(* Logix 5000 project; controller OCV_Tester_EnSG vendor 1 type 14 code 106 rev 32.11; software revision 32.02 *)

TASK MainTask (continuous, watchdog 500 ms) : MainProgram

MODULES
   Local : vendor 1 type 14 code 106 (Compact 0, rev 32.11)
      DI_H2 : vendor 1 type 7 code 69 (Compact 2, rev 3.1, Input RPI 0.5 ms)
      DI_H : vendor 1 type 7 code 69 (Compact 1, rev 3.1, Input RPI 0.5 ms)
      AI : 1769-IF8 (Compact 4, rev 1.1, Output RPI 1 ms)
      DOut : vendor 1 type 7 code 73 (Compact 3, rev 3.1, Output RPI 1 ms)
      AI2 : vendor 1 type 10 code 46 (Compact 5, rev 1.1, Output RPI 1 ms)
      CPU : vendor 1 type 14 code 156 (Ethernet 172.20.7.50, rev 32.1)
      ConveyorMot : PowerFlex 525-EENET (Ethernet 172.20.9.12, rev 5.2, Output RPI 20 ms)
END_MODULES

VAR_GLOBAL   (* controller tags *)
   alwaysOK : BOOL; {constant}
   Angle : DINT := 229;
   AngleCal : DINT := 229;
   AngleOffset : DINT;
   AngleRaw : DINT := 131;   // encoder angle
   Auto : BOOL := 1;
   AVE_NOK_Control : CONTROL := (LEN := 20);
   battMon : DINT[20] := ([0] := 1552, [2] := 1641, [3] := 2222, [4] := 935, [5] := 1318, [6] := 1513, [7] := 1473, [8] := 1630, [9] := 951, [10] := 1594, [12] := 1605);
   battV : DINT[64] := ([0] := 1600, [1] := 1600, [2] := 1600, [3] := 1600, [4] := 1600, [5] := 1600, [6] := 1600, [7] := 1600, [8] := 1600, [9] := 1600, [10] := 1600, [11] := 1600, [12] := 1600, [13] := 1600, [14] := 1600, [15] := 1600, [16] := 1600, [17] := 1600, [18] := 1600, [19] := 1600, [20] := 1600, [21] := 1600, [22] := 1600, [23] := 1600, [24] := 1600, [25] := 1600, [26] := 1600, [27] := 1600, [28] := 1600, [29] := 1600, [30] := 1600, [31] := 1600, [32] := 1600, [33] := 1600, [34] := 1600, [35] := 1600, [36] := 1600, [37] := 1600, [38] := 1600, [39] := 1600, [40] := 1600, [41] := 1600, [42] := 1600, [43] := 1600, [44] := 1600, [45] := 1600, [46] := 1600, [47] := 1600, [48] := 1600, [49] := 1600, [50] := 1600, [51] := 1600, [52] := 1600, [53] := 1600, [54] := 1600, [55] := 1600, [56] := 1600, [57] := 1600, [58] := 1600, [59] := 1600,
        [60] := 1600, [61] := 1600, [62] := 1600, [63] := 1600);
   battV_NOK : INT[21] := ([0] := 1491, [1] := 1491, [2] := 1491, [3] := 1491, [4] := 1491, [5] := 1491, [6] := 1491, [7] := 1491, [8] := 1491, [9] := 1491, [10] := 1491, [11] := 1491, [12] := 1491, [13] := 1491, [14] := 1491, [15] := 1491, [16] := 1491, [17] := 1491, [18] := 1491, [19] := 1491);
   battV_NOK_avg : DINT := -25;
   blink1s : BOOL;
   blower0 : BOOL;
   cal_curVoltRaw : INT;
   cal_nom : INT := 2000; {constant}
   cal_T : DINT;
   cal_timeTOFPre : REAL := 0.25;
   cal_TimeTONPre : INT := 79;
   contact_dur_t : TIMER[20] := ([0].PRE := 2147483645, [0].ACC := 1742075, [1].PRE := 2147483645, [1].ACC := 1742075, [2].PRE := 2147483645, [2].ACC := 1742075, [3].PRE := 2147483645, [3].ACC := 1742075, [4].PRE := 2147483645, [4].ACC := 1742075, [5].PRE := 2147483645, [5].ACC := 1742075, [6].PRE := 2147483645, [6].ACC := 1742075, [7].PRE := 2147483645, [7].ACC := 1742075);
   cutOff_thrs : INT := 1597;
   d_idx : INT;
   DataV : INT[20] := ([0] := 1491, [1] := 1895, [2] := 1628, [4] := 1650, [5] := 1609, [6] := 1467, [7] := 1634, [8] := 1648, [9] := 1407, [11] := 1563, [12] := 969, [13] := 1519, [14] := 1641, [15] := 1050, [16] := 1692, [17] := 1604, [18] := 1643, [19] := 1572);
   defects : DINT[5] := ([0] := 536870911, [1] := 4324957);
   dummy3 : BOOL;
   dummy4 : BOOL;
   dummy5 : BOOL;
   eStop : BOOL;
   even : BOOL;
   fail_ejectSerp : BOOL := 1;
   fail_ejectValidation : BOOL;
   failed : BOOL[32];
   FailToRemove : BOOL := 1;   // Failed to remove battery
   Fault : BOOL;
   fault_jam : BOOL;
   FFOMonCtrl : CONTROL := (LEN := 20, POS := 19);
   FFONOKCtrl : CONTROL := (LEN := 21, POS := 20);
   FFOPrbNOKCtrl : CONTROL := (LEN := 21, POS := 20);
   FloatMode : BOOL;
   hmi_accept_thrs : INT := 1600;
   hmi_blower0 : BOOL;
   hmi_blower1 : BOOL;
   hmi_calMax : BOOL[32];
   hmi_calMin : BOOL[32];
   hmi_clearFault : BOOL;
   hmi_contactDur : DINT[20] := ([0] := 457, [1] := 1096, [2] := 2008, [3] := 182, [4] := 1187, [5] := 456, [6] := 457, [7] := 1096, [8] := 182, [9] := 273, [10] := 457, [11] := 1095, [12] := 2008, [13] := 182, [14] := 1187, [15] := 456, [16] := 457, [17] := 1096, [18] := 182, [19] := 273);   // Contact Duration
   hmi_delta : INT := 3;   // float test delta mV
   hmi_jog : BOOL;
   hmi_setSpeedRef : INT := 45;   // HMI_SetSpeed
   hmi_settingSave : BOOL;
   hmi_startingVolt : DINT := 1600;   // Init Buffer val
   i : INT;
   idx : DINT := 64;
   infeed_start_pre : INT;
   infeed_stop_pre : INT;
   lastVolt2 : DINT;
   motJam_t : DINT := 2000;   // Motor Jam T Threshold
   MotStart : BOOL;
   nc_ps_output : BOOL;
   nc_safetyContAux : BOOL;
   nofBatt : DINT := 18562;   // Number of Battery tested
   nofFailBatt : DINT := 906;
   NOK : BOOL;
   NOKK : BOOL;
   odd : BOOL;
   ons1 : DINT := 1073758208;
   Paused : BOOL;
   pb_Emergency : BOOL;
   pb_Start : BOOL;
   pb_Stop : BOOL;
   press_switch : BOOL := 1;
   probeId_NOK : INT[21] := ([0] := 1, [1] := 1, [2] := 1, [3] := 1, [4] := 1, [5] := 1, [6] := 1, [7] := 1, [8] := 1, [9] := 1, [10] := 1, [11] := 1, [12] := 1, [13] := 1, [14] := 1, [15] := 1, [16] := 1, [17] := 1, [18] := 1, [19] := 1);
   probeIdx : INT := 14;   // probe index
   ps_ejectSerp : BOOL := 1;
   ps_exist : BOOL;
   ps_index : BOOL;
   ps_inFeed : BOOL := 1;   // serpentine top
   ps_verify : BOOL;   // to verify a success remove
   ps_wheel : BOOL := 1;
   Reset : BOOL;
   Run : BOOL;
   safety_sys_ok : BOOL;
   speed : DINT;   // battery per minute
   Start : BOOL;   // Start State
   sw_door : BOOL;
   sw_doorSide : BOOL;   // Door Switch Side
   sw_doorTop : BOOL;
   timeTOFPre : DINT;
   tmr_blower0_en : BOOL;
   tmr_infeed : TIMER := (PRE := 2000);
   unloadBattV_NOK : DINT := 1491;
   unloadedBattMon : DINT := 1644;
   unloadProbe_NOK : INT := 1;
   use_calVal : BOOL;
   V_min : INT := 200;   // detect batt V
   v_rampThrs : INT := 1650;
   VMax : INT[20];
   VMin : INT[20];
   volt : INT[20];
   warning : BOOL;
   warningLamp : BOOL;
END_VAR

PROGRAM MainProgram   (* main routine MainRoutine *)
VAR
   _blower1TmrPre_tot : DINT;
   _blowerTmrPre : DINT := 130;
   _blowerTmrPre_tot : DINT := -20;
   _oddEvenRest : INT;
   AngleLimit : DINT[21] := ([0] := 340, [1] := 358, [2] := 16, [3] := 34, [4] := 52, [5] := 70, [6] := 88, [7] := 106, [8] := 124, [9] := 142, [10] := 160, [11] := 178, [12] := 196, [13] := 214, [14] := 232, [15] := 250, [16] := 268, [17] := 286, [18] := 304, [19] := 322, [20] := 340);
   AVE_Control : CONTROL := (LEN := 64);   // battery average ctrl
   battCnt : COUNTER;
   battV_avg : DINT := 1600;   // battery voltage average
   blower0_tof_pre : DINT;
   blower_react_ms : DINT := 20;
   BSLCtrl : CONTROL := (LEN := 64);
   buf_battVLen : INT := 64;   // buffer length 64
   calcSpeed : BOOL;
   clearFFO : BOOL;
   contact_Idx : INT;
   contact_t : TIMER[20] := ([0].PRE := 2147483647, [1].PRE := 2147483647, [2].PRE := 2147483647, [3].PRE := 2147483647, [4].PRE := 2147483647, [5].PRE := 2147483647, [6].PRE := 2147483647, [7].PRE := 2147483647, [8].PRE := 2147483647, [9].PRE := 2147483647, [10].PRE := 2147483647, [11].PRE := 2147483647, [12].PRE := 2147483647, [13].PRE := 2147483647, [14].PRE := 2147483647, [15].PRE := 2147483647, [16].PRE := 2147483647, [17].PRE := 2147483647, [18].PRE := 2147483647, [19].PRE := 2147483647);
   contactDur_t : TIMER[20];
   Data1 : DINT;
   dbc_tof : TIMER[2] := ([0].PRE := 2, [0].EN := 1, [0].DN := 1);
   dbc_ton : TIMER[2] := ([0].PRE := 2, [0].ACC := 3, [0].EN := 1, [0].DN := 1);
   DelayBlow : BOOL;
   deltaNofBatt : DINT;
   deltaTSpeed : DINT;
   dummyProbeEn : BOOL;
   en_blower : BOOL := 1;
   enableDummyPsIndex : BOOL;
   Failed : BOOL;
   FFOCtrl : CONTROL := (LEN := 60, POS := 60, DN := 1);
   FFOCtrl_defects : CONTROL;
   fifo : DINT;
   ForVIdx : DINT := 11;
   freeTmr : TIMER := (PRE := 2147483646, ACC := 138932, EN := 1, TT := 1);
   hmi_rev : BOOL := 1;
   hmi_setAngle0 : BOOL;   // set Offset Angle 0
   hmi_setSpeedRef100 : INT := 4500;   // hmi_setSpeedRef*100
   index : BOOL;
   lastScan : DINT := 138932;
   lastVolt : DINT;
   MaxV : INT[20] := ([1] := 1895, [2] := 1619, [3] := 1635, [4] := 1543, [5] := 1170, [8] := 287);
   nofBattOld : DINT;
   OK : BOOL := 1;
   ons : INT;
   ons2 : DINT := 68;
   Passed : BOOL;
   pb_DoorSw : BOOL;
   pb_SafetyRst : BOOL;   // pb safety reset
   ps_exist_ons : BOOL;
   px_inFeed : BOOL;   // serpentine top
   Safety : BOOL;
   StartAngle : DINT := 340;
   startContact_ts : DINT[20] := ([0] := 138649, [1] := 138887, [2] := 138808, [3] := 138887, [4] := 98255);   // Contact start
   TimeTONPre : DINT := -79;
   tmr_blower0 : TIMER := (PRE := 229);
   tmr_blower0_en : BOOL;
   tmr_blower0_TOF : TIMER := (PRE := 77);
   tmr_infeed_start : TIMER := (PRE := 1700, EN := 1, DN := 1);
   tmr_infeed_stop : TIMER := (PRE := 250);
   TmrDuration : TIMER := (PRE := 2147483647);
   tof1s : TIMER := (TT := 1, DN := 1);
   ton1s : TIMER;
   ton_blower0 : DINT;
   unloadBattV : DINT;   // unloaded battV element array
   unloadFFODefects : DINT;   // unloaded defects fifo element
END_VAR

ROUTINE _00_Diagnostics   (* ladder *)
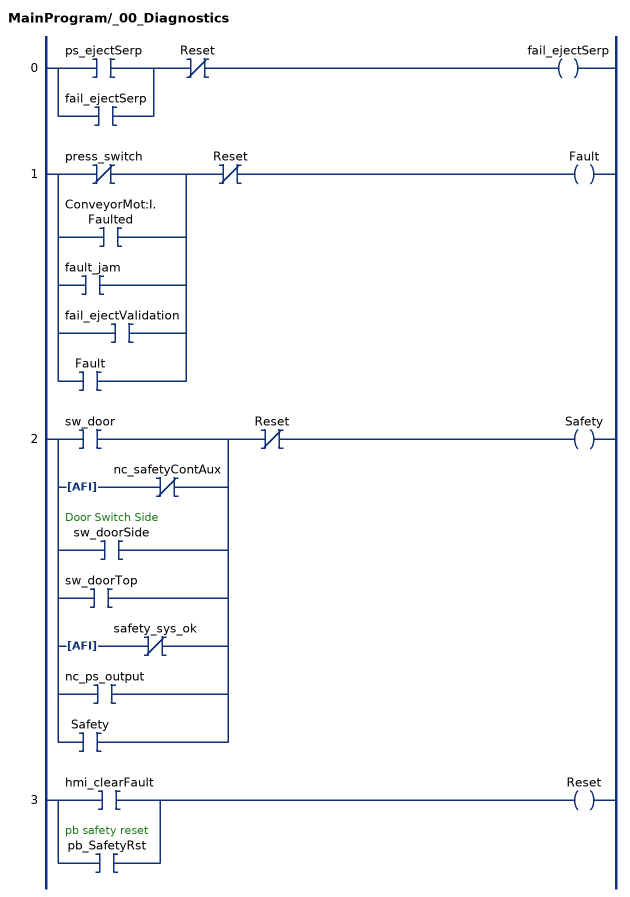
   0: [XIC(ps_ejectSerp) ,XIC(fail_ejectSerp) ]XIO(Reset)OTE(fail_ejectSerp);
   1: [XIO(press_switch) ,XIC(ConveyorMot:I.Faulted) ,XIC(fault_jam) ,XIC(fail_ejectValidation) ,XIC(Fault) ]XIO(Reset)OTE(Fault);
   2: [XIC(sw_door) ,AFI() XIO(nc_safetyContAux) ,XIC(sw_doorSide) ,XIC(sw_doorTop) ,AFI() XIO(safety_sys_ok) ,XIC(nc_ps_output) ,XIC(Safety) ]XIO(Reset)OTE(Safety);
   3: [XIC(hmi_clearFault) ,XIC(pb_SafetyRst) ]OTE(Reset);
END_ROUTINE

ROUTINE _01_Inputs   (* ladder *)
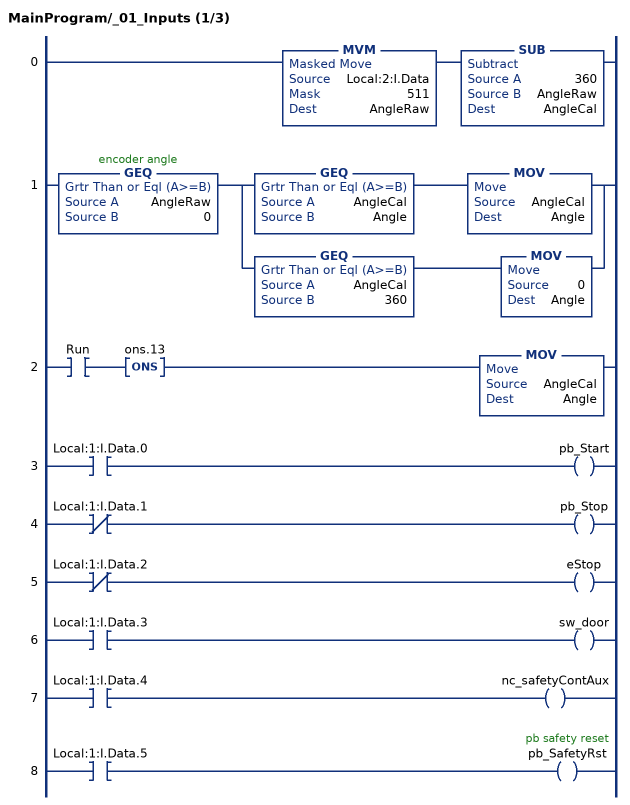
   0: MVM(Local:2:I.Data,511,AngleRaw)SUB(360,AngleRaw,AngleCal);
   1: GEQ(AngleRaw,0)[GEQ(AngleCal,Angle) MOV(AngleCal,Angle) ,GEQ(AngleCal,360) MOV(0,Angle) ];
   2: XIC(Run)ONS(ons.13)MOV(AngleCal,Angle);
   3: XIC(Local:1:I.Data.0)OTE(pb_Start);
   4: XIO(Local:1:I.Data.1)OTE(pb_Stop);
   5: XIO(Local:1:I.Data.2)OTE(eStop);
   6: XIC(Local:1:I.Data.3)OTE(sw_door);
   7: XIC(Local:1:I.Data.4)OTE(nc_safetyContAux);
   8: XIC(Local:1:I.Data.5)OTE(pb_SafetyRst);
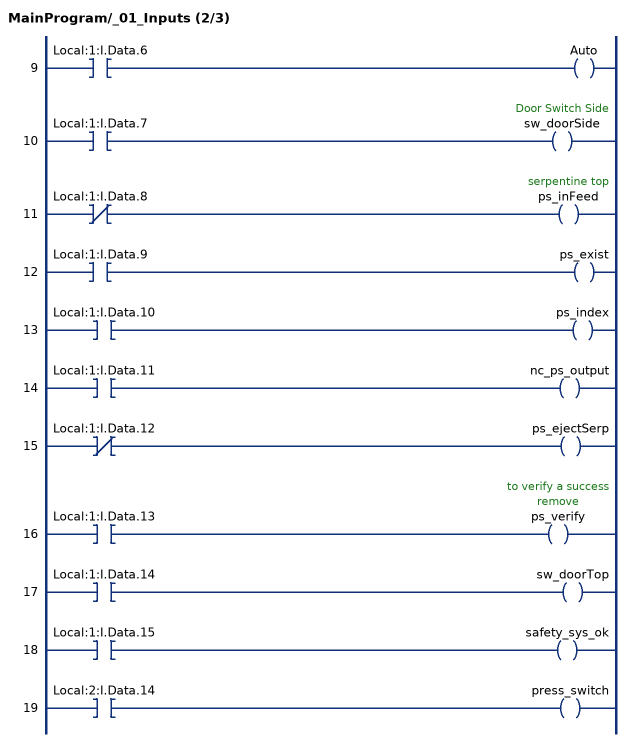
   9: XIC(Local:1:I.Data.6)OTE(Auto);
   10: XIC(Local:1:I.Data.7)OTE(sw_doorSide);
   11: XIO(Local:1:I.Data.8)OTE(ps_inFeed);
   12: XIC(Local:1:I.Data.9)OTE(ps_exist);
   13: XIC(Local:1:I.Data.10)OTE(ps_index);
   14: XIC(Local:1:I.Data.11)OTE(nc_ps_output);
   15: XIO(Local:1:I.Data.12)OTE(ps_ejectSerp);
   16: XIC(Local:1:I.Data.13)OTE(ps_verify);
   17: XIC(Local:1:I.Data.14)OTE(sw_doorTop);
   18: XIC(Local:1:I.Data.15)OTE(safety_sys_ok);
   19: XIC(Local:2:I.Data.14)OTE(press_switch);
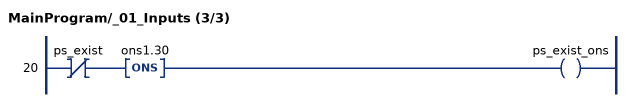
   20: XIO(ps_exist)ONS(ons1.30)OTE(ps_exist_ons);
END_ROUTINE

ROUTINE _02_Run   (* ladder *)
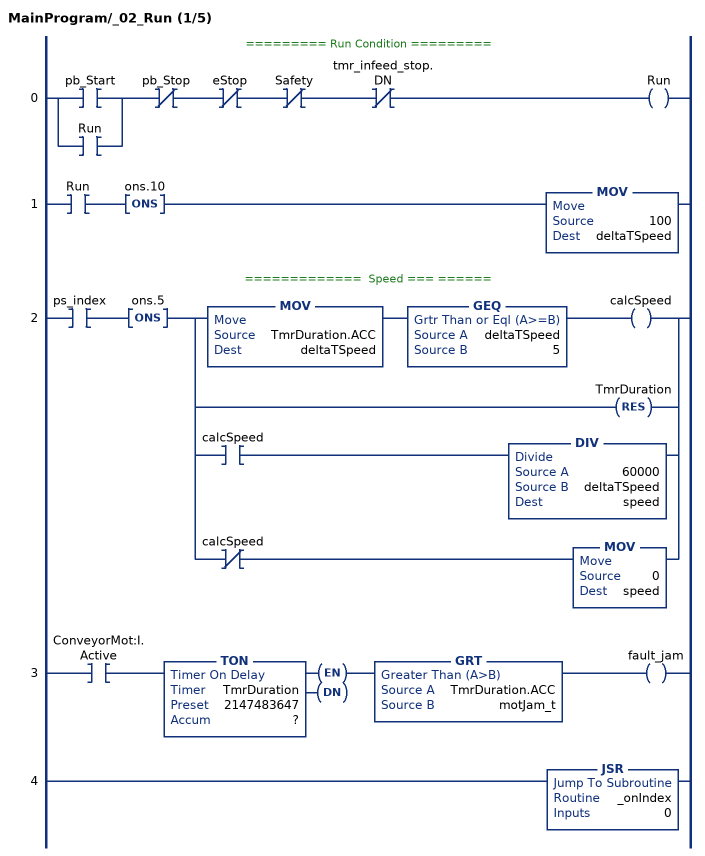
   // ========= Run Condition =========
   0: [XIC(pb_Start) ,XIC(Run) ]XIO(pb_Stop)XIO(eStop)XIO(Safety)XIO(tmr_infeed_stop.DN)OTE(Run);
   1: XIC(Run)ONS(ons.10)MOV(100,deltaTSpeed);
   // =============  Speed === ======
   2: XIC(ps_index)ONS(ons.5)[MOV(TmrDuration.ACC,deltaTSpeed) GEQ(deltaTSpeed,5) OTE(calcSpeed) ,RES(TmrDuration) ,XIC(calcSpeed) DIV(60000,deltaTSpeed,speed) ,XIO(calcSpeed) MOV(0,speed) ];
   3: XIC(ConveyorMot:I.Active)TON(TmrDuration,?,?)GRT(TmrDuration.ACC,motJam_t)OTE(fault_jam);
   4: JSR(_onIndex,0);
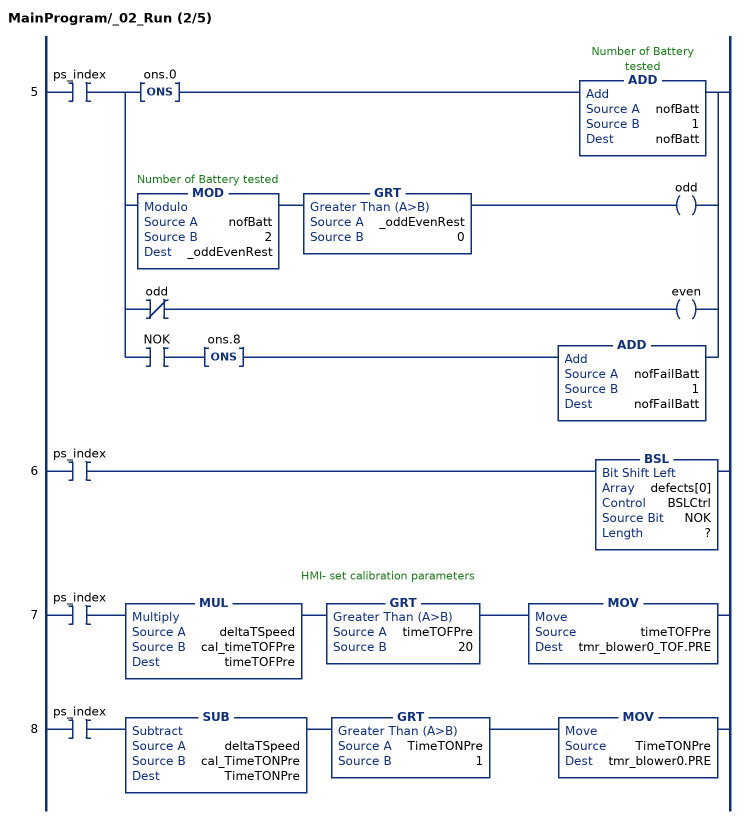
   5: XIC(ps_index)[ONS(ons.0) ADD(nofBatt,1,nofBatt) ,MOD(nofBatt,2,_oddEvenRest) GRT(_oddEvenRest,0) OTE(odd) ,XIO(odd) OTE(even) ,XIC(NOK) ONS(ons.8) ADD(nofFailBatt,1,nofFailBatt) ];
   6: XIC(ps_index)BSL(defects[0],BSLCtrl,NOK,?);
   // HMI- set calibration parameters
   7: XIC(ps_index)MUL(deltaTSpeed,cal_timeTOFPre,timeTOFPre)GRT(timeTOFPre,20)MOV(timeTOFPre,tmr_blower0_TOF.PRE);
   8: XIC(ps_index)SUB(deltaTSpeed,cal_TimeTONPre,TimeTONPre)GRT(TimeTONPre,1)MOV(TimeTONPre,tmr_blower0.PRE);
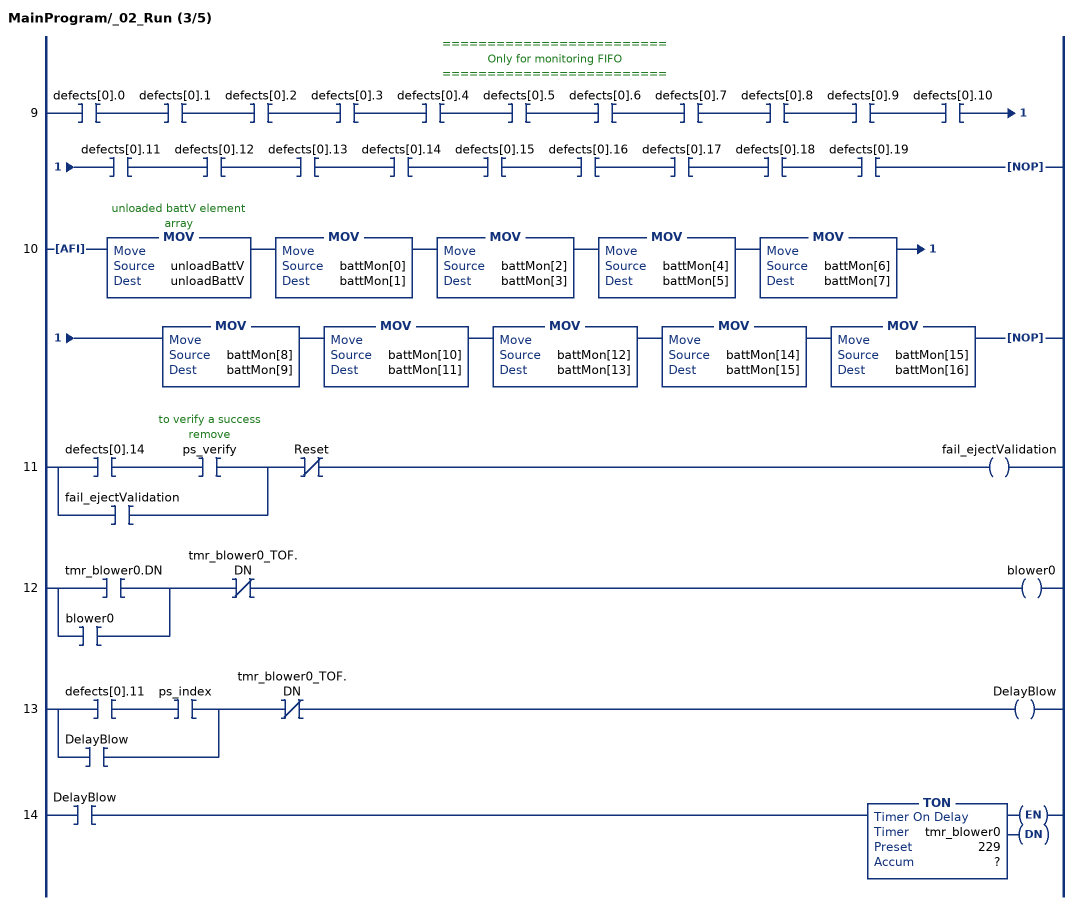
   // =========================
   // Only for monitoring FIFO
   // =========================
   9: XIC(defects[0].0)XIC(defects[0].1)XIC(defects[0].2)XIC(defects[0].3)XIC(defects[0].4)XIC(defects[0].5)XIC(defects[0].6)XIC(defects[0].7)XIC(defects[0].8)XIC(defects[0].9)XIC(defects[0].10)XIC(defects[0].11)XIC(defects[0].12)XIC(defects[0].13)XIC(defects[0].14)XIC(defects[0].15)XIC(defects[0].16)XIC(defects[0].17)XIC(defects[0].18)XIC(defects[0].19)NOP();
   10: AFI()MOV(unloadBattV,unloadBattV)MOV(battMon[0],battMon[1])MOV(battMon[2],battMon[3])MOV(battMon[4],battMon[5])MOV(battMon[6],battMon[7])MOV(battMon[8],battMon[9])MOV(battMon[10],battMon[11])MOV(battMon[12],battMon[13])MOV(battMon[14],battMon[15])MOV(battMon[15],battMon[16])NOP();
   11: [XIC(defects[0].14) XIC(ps_verify) ,XIC(fail_ejectValidation) ]XIO(Reset)OTE(fail_ejectValidation);
   12: [XIC(tmr_blower0.DN) ,XIC(blower0) ]XIO(tmr_blower0_TOF.DN)OTE(blower0);
   13: [XIC(defects[0].11) XIC(ps_index) ,XIC(DelayBlow) ]XIO(tmr_blower0_TOF.DN)OTE(DelayBlow);
   14: XIC(DelayBlow)TON(tmr_blower0,?,?);
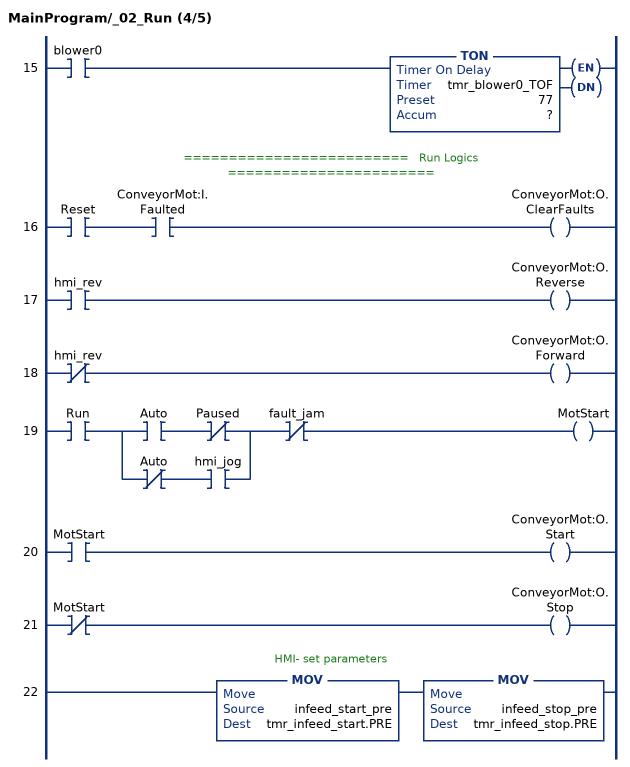
   15: XIC(blower0)TON(tmr_blower0_TOF,?,?);
   // =========================   Run Logics   =======================
   16: XIC(Reset)XIC(ConveyorMot:I.Faulted)OTE(ConveyorMot:O.ClearFaults);
   17: XIC(hmi_rev)OTE(ConveyorMot:O.Reverse);
   18: XIO(hmi_rev)OTE(ConveyorMot:O.Forward);
   19: XIC(Run)[XIC(Auto) XIO(Paused) ,XIO(Auto) XIC(hmi_jog) ]XIO(fault_jam)OTE(MotStart);
   20: XIC(MotStart)OTE(ConveyorMot:O.Start);
   21: XIO(MotStart)OTE(ConveyorMot:O.Stop);
   // HMI- set parameters
   22: MOV(infeed_start_pre,tmr_infeed_start.PRE)MOV(infeed_stop_pre,tmr_infeed_stop.PRE);
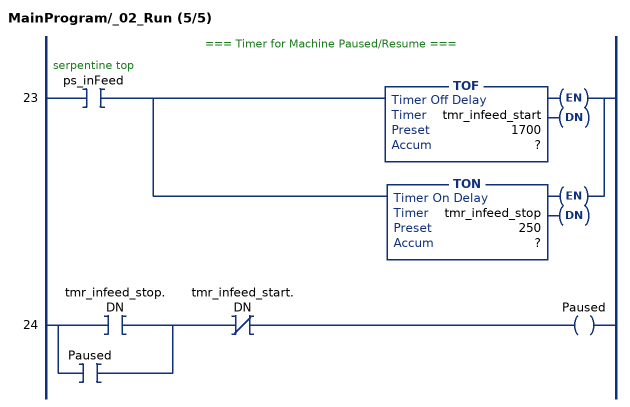
   // === Timer for Machine Paused/Resume ===
   23: XIC(ps_inFeed)[TOF(tmr_infeed_start,?,?) ,TON(tmr_infeed_stop,?,?) ];
   24: [XIC(tmr_infeed_stop.DN) ,XIC(Paused) ]XIO(tmr_infeed_start.DN)OTE(Paused);
END_ROUTINE

ROUTINE _03_Angle   (* ladder *)
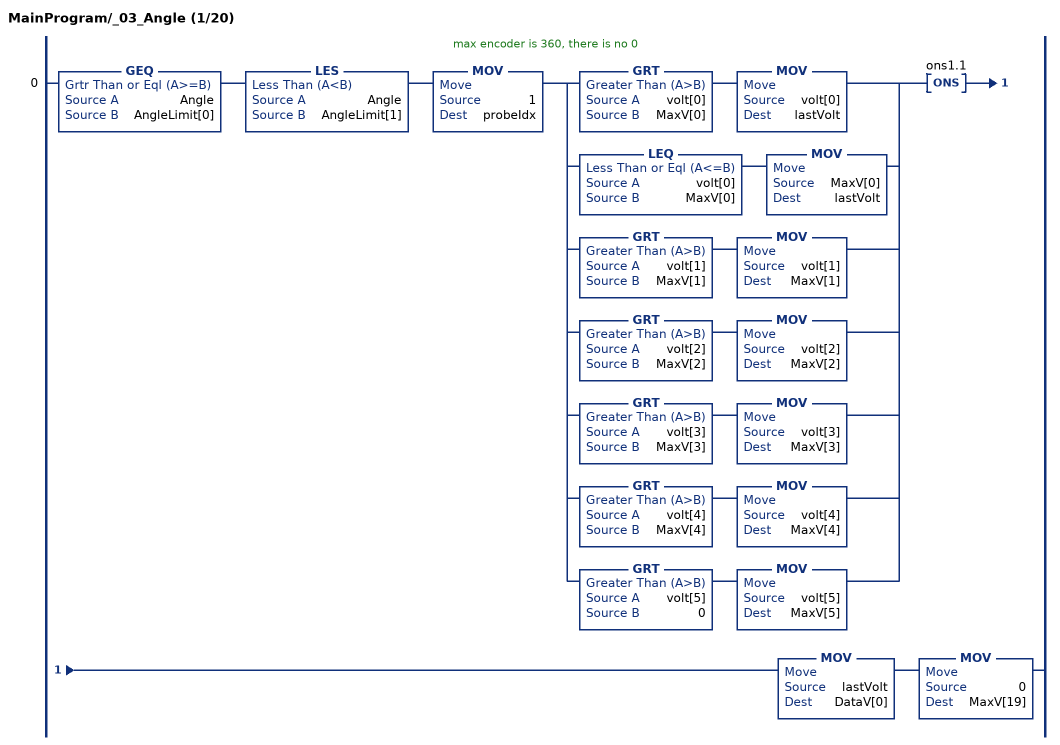
   // max encoder is 360, there is no 0
   0: GEQ(Angle,AngleLimit[0])LES(Angle,AngleLimit[1])MOV(1,probeIdx)[GRT(volt[0],MaxV[0]) MOV(volt[0],lastVolt) ,LEQ(volt[0],MaxV[0]) MOV(MaxV[0],lastVolt) ,GRT(volt[1],MaxV[1]) MOV(volt[1],MaxV[1]) ,GRT(volt[2],MaxV[2]) MOV(volt[2],MaxV[2]) ,GRT(volt[3],MaxV[3]) MOV(volt[3],MaxV[3]) ,GRT(volt[4],MaxV[4]) MOV(volt[4],MaxV[4]) ,GRT(volt[5],0) MOV(volt[5],MaxV[5]) ]ONS(ons1.1)MOV(lastVolt,DataV[0])MOV(0,MaxV[19]);
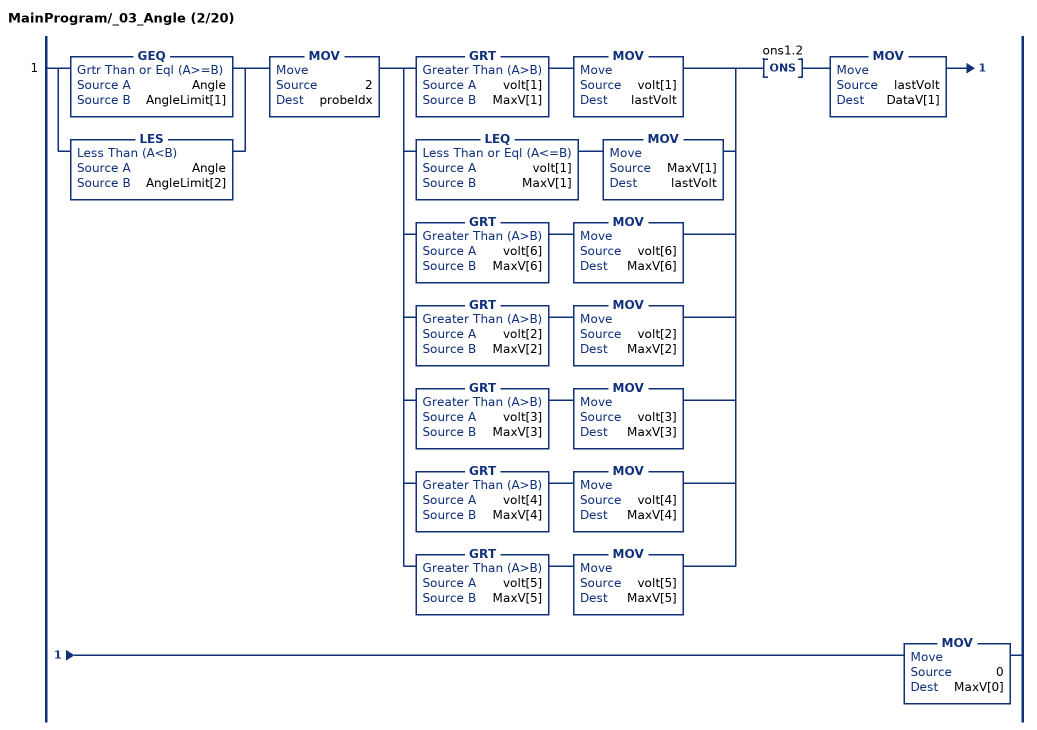
   1: [GEQ(Angle,AngleLimit[1]) ,LES(Angle,AngleLimit[2]) ]MOV(2,probeIdx)[GRT(volt[1],MaxV[1]) MOV(volt[1],lastVolt) ,LEQ(volt[1],MaxV[1]) MOV(MaxV[1],lastVolt) ,GRT(volt[6],MaxV[6]) MOV(volt[6],MaxV[6]) ,GRT(volt[2],MaxV[2]) MOV(volt[2],MaxV[2]) ,GRT(volt[3],MaxV[3]) MOV(volt[3],MaxV[3]) ,GRT(volt[4],MaxV[4]) MOV(volt[4],MaxV[4]) ,GRT(volt[5],MaxV[5]) MOV(volt[5],MaxV[5]) ]ONS(ons1.2)MOV(lastVolt,DataV[1])MOV(0,MaxV[0]);
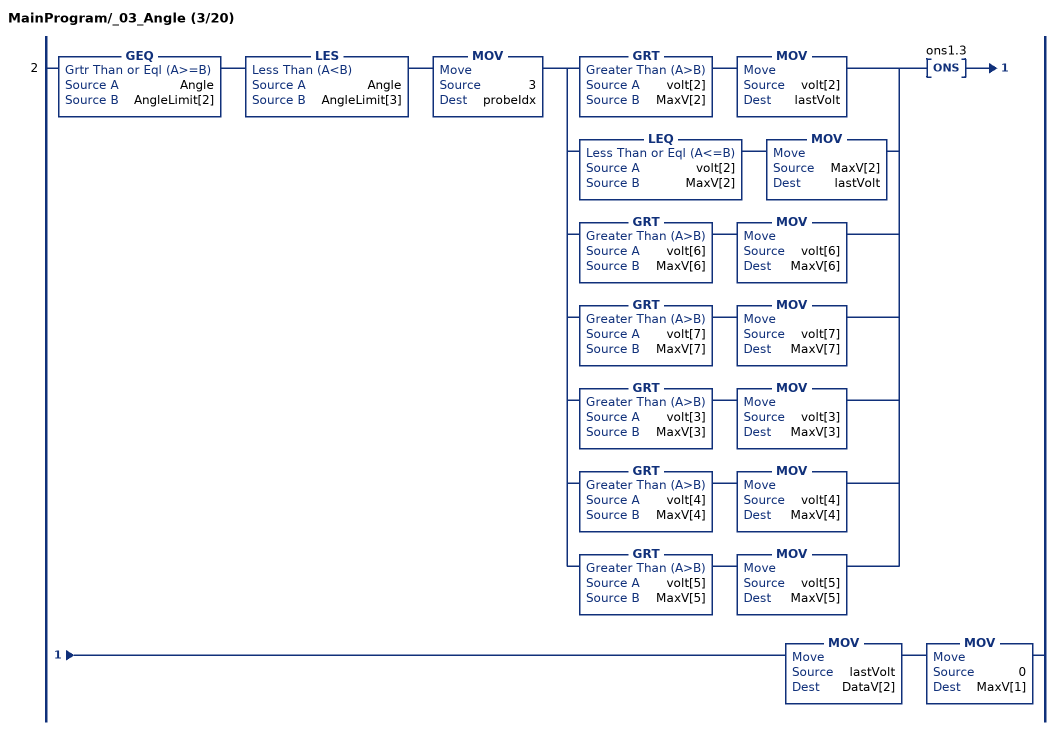
   2: GEQ(Angle,AngleLimit[2])LES(Angle,AngleLimit[3])MOV(3,probeIdx)[GRT(volt[2],MaxV[2]) MOV(volt[2],lastVolt) ,LEQ(volt[2],MaxV[2]) MOV(MaxV[2],lastVolt) ,GRT(volt[6],MaxV[6]) MOV(volt[6],MaxV[6]) ,GRT(volt[7],MaxV[7]) MOV(volt[7],MaxV[7]) ,GRT(volt[3],MaxV[3]) MOV(volt[3],MaxV[3]) ,GRT(volt[4],MaxV[4]) MOV(volt[4],MaxV[4]) ,GRT(volt[5],MaxV[5]) MOV(volt[5],MaxV[5]) ]ONS(ons1.3)MOV(lastVolt,DataV[2])MOV(0,MaxV[1]);
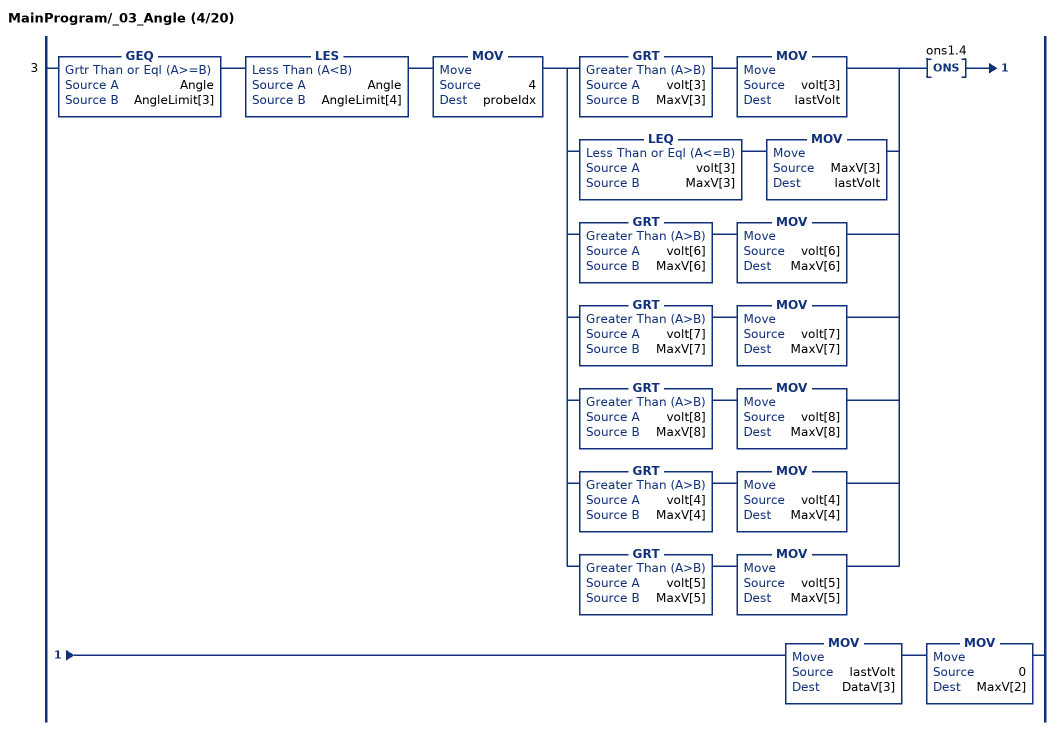
   3: GEQ(Angle,AngleLimit[3])LES(Angle,AngleLimit[4])MOV(4,probeIdx)[GRT(volt[3],MaxV[3]) MOV(volt[3],lastVolt) ,LEQ(volt[3],MaxV[3]) MOV(MaxV[3],lastVolt) ,GRT(volt[6],MaxV[6]) MOV(volt[6],MaxV[6]) ,GRT(volt[7],MaxV[7]) MOV(volt[7],MaxV[7]) ,GRT(volt[8],MaxV[8]) MOV(volt[8],MaxV[8]) ,GRT(volt[4],MaxV[4]) MOV(volt[4],MaxV[4]) ,GRT(volt[5],MaxV[5]) MOV(volt[5],MaxV[5]) ]ONS(ons1.4)MOV(lastVolt,DataV[3])MOV(0,MaxV[2]);
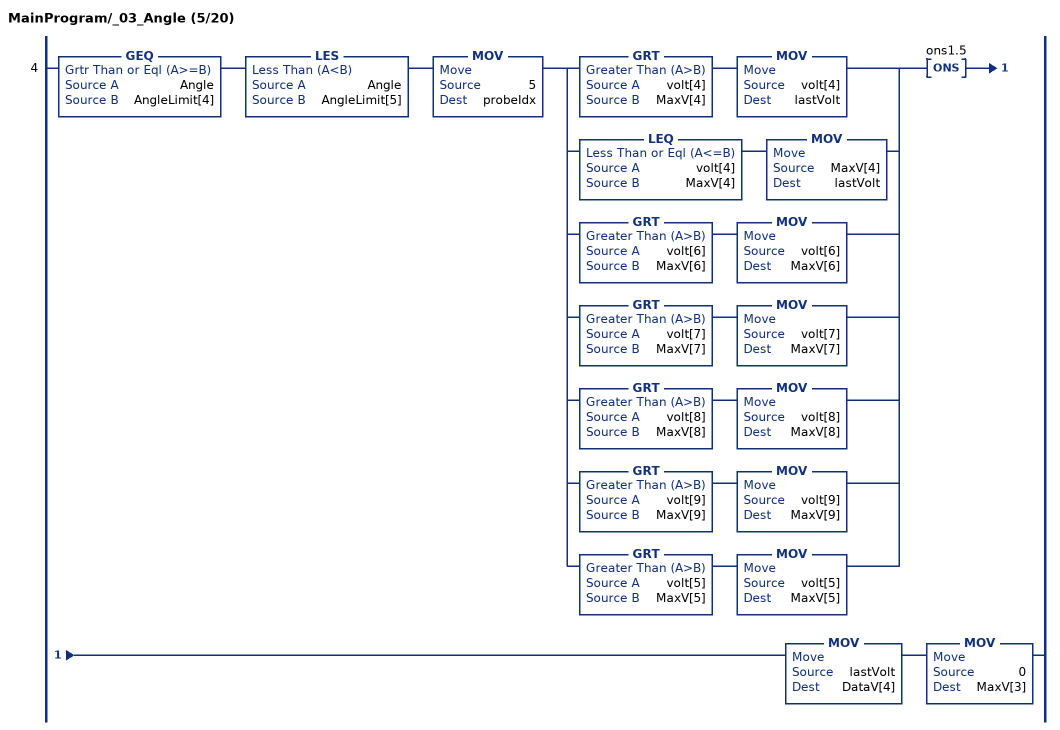
   4: GEQ(Angle,AngleLimit[4])LES(Angle,AngleLimit[5])MOV(5,probeIdx)[GRT(volt[4],MaxV[4]) MOV(volt[4],lastVolt) ,LEQ(volt[4],MaxV[4]) MOV(MaxV[4],lastVolt) ,GRT(volt[6],MaxV[6]) MOV(volt[6],MaxV[6]) ,GRT(volt[7],MaxV[7]) MOV(volt[7],MaxV[7]) ,GRT(volt[8],MaxV[8]) MOV(volt[8],MaxV[8]) ,GRT(volt[9],MaxV[9]) MOV(volt[9],MaxV[9]) ,GRT(volt[5],MaxV[5]) MOV(volt[5],MaxV[5]) ]ONS(ons1.5)MOV(lastVolt,DataV[4])MOV(0,MaxV[3]);
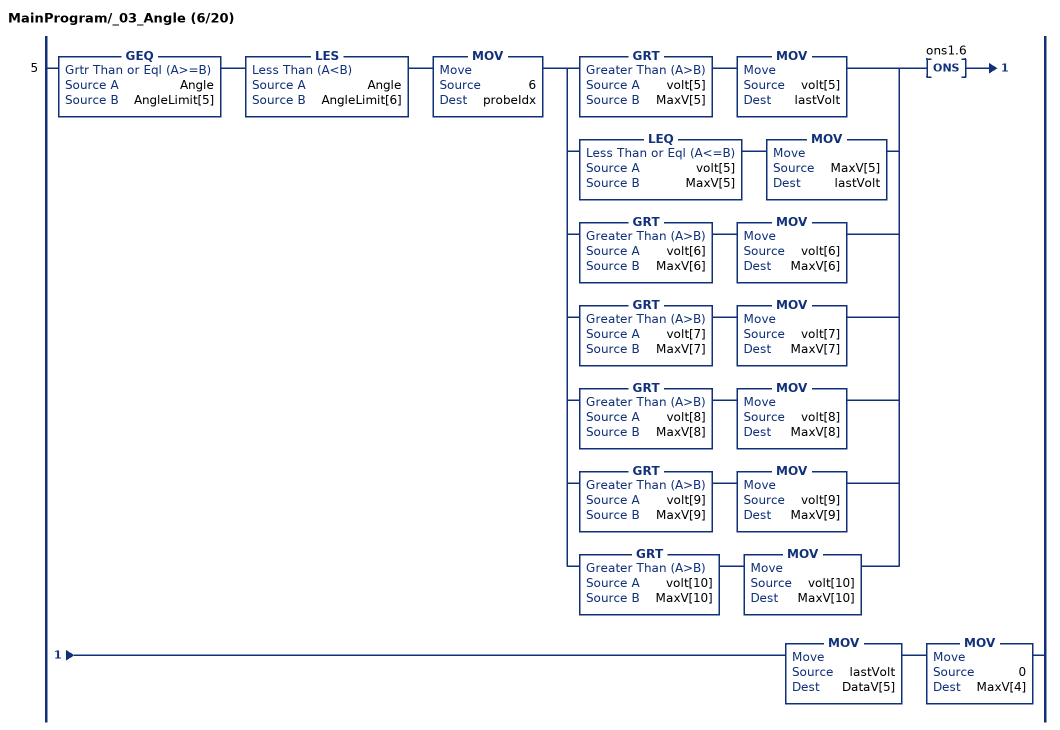
   5: GEQ(Angle,AngleLimit[5])LES(Angle,AngleLimit[6])MOV(6,probeIdx)[GRT(volt[5],MaxV[5]) MOV(volt[5],lastVolt) ,LEQ(volt[5],MaxV[5]) MOV(MaxV[5],lastVolt) ,GRT(volt[6],MaxV[6]) MOV(volt[6],MaxV[6]) ,GRT(volt[7],MaxV[7]) MOV(volt[7],MaxV[7]) ,GRT(volt[8],MaxV[8]) MOV(volt[8],MaxV[8]) ,GRT(volt[9],MaxV[9]) MOV(volt[9],MaxV[9]) ,GRT(volt[10],MaxV[10]) MOV(volt[10],MaxV[10]) ]ONS(ons1.6)MOV(lastVolt,DataV[5])MOV(0,MaxV[4]);
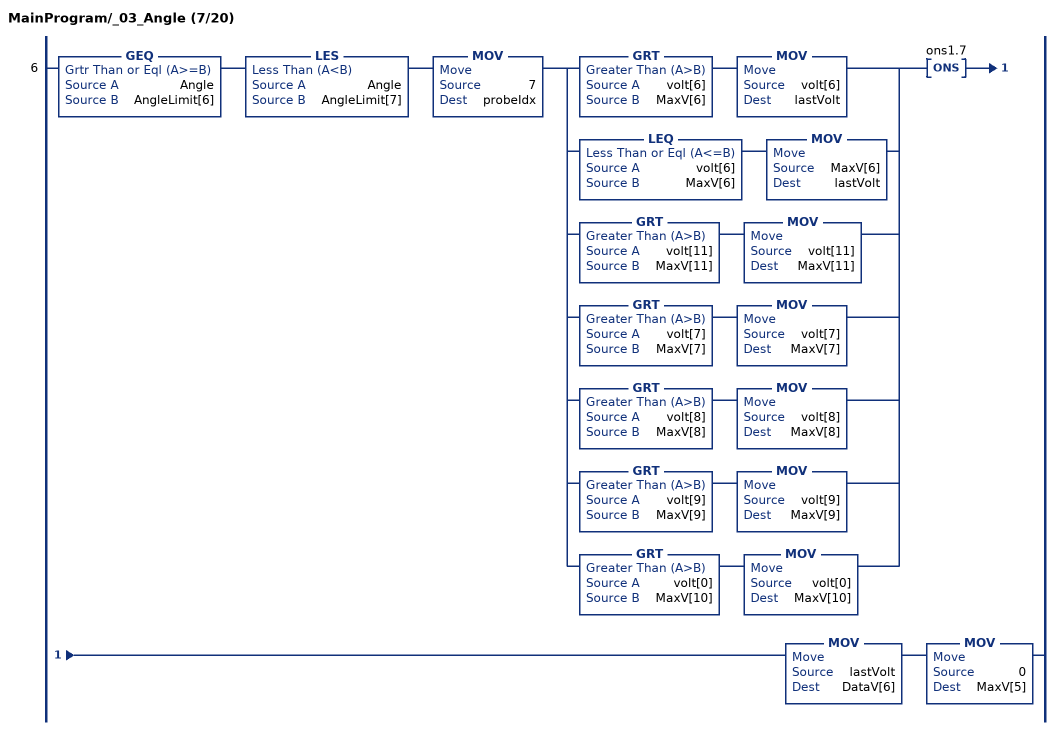
   6: GEQ(Angle,AngleLimit[6])LES(Angle,AngleLimit[7])MOV(7,probeIdx)[GRT(volt[6],MaxV[6]) MOV(volt[6],lastVolt) ,LEQ(volt[6],MaxV[6]) MOV(MaxV[6],lastVolt) ,GRT(volt[11],MaxV[11]) MOV(volt[11],MaxV[11]) ,GRT(volt[7],MaxV[7]) MOV(volt[7],MaxV[7]) ,GRT(volt[8],MaxV[8]) MOV(volt[8],MaxV[8]) ,GRT(volt[9],MaxV[9]) MOV(volt[9],MaxV[9]) ,GRT(volt[0],MaxV[10]) MOV(volt[0],MaxV[10]) ]ONS(ons1.7)MOV(lastVolt,DataV[6])MOV(0,MaxV[5]);
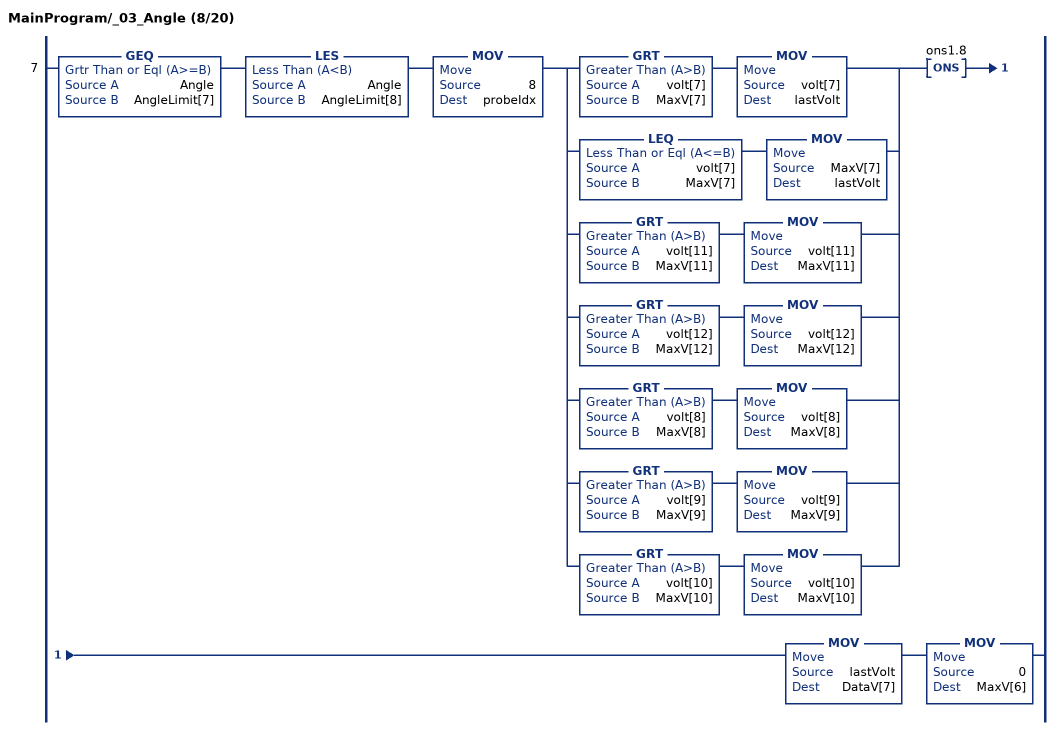
   7: GEQ(Angle,AngleLimit[7])LES(Angle,AngleLimit[8])MOV(8,probeIdx)[GRT(volt[7],MaxV[7]) MOV(volt[7],lastVolt) ,LEQ(volt[7],MaxV[7]) MOV(MaxV[7],lastVolt) ,GRT(volt[11],MaxV[11]) MOV(volt[11],MaxV[11]) ,GRT(volt[12],MaxV[12]) MOV(volt[12],MaxV[12]) ,GRT(volt[8],MaxV[8]) MOV(volt[8],MaxV[8]) ,GRT(volt[9],MaxV[9]) MOV(volt[9],MaxV[9]) ,GRT(volt[10],MaxV[10]) MOV(volt[10],MaxV[10]) ]ONS(ons1.8)MOV(lastVolt,DataV[7])MOV(0,MaxV[6]);
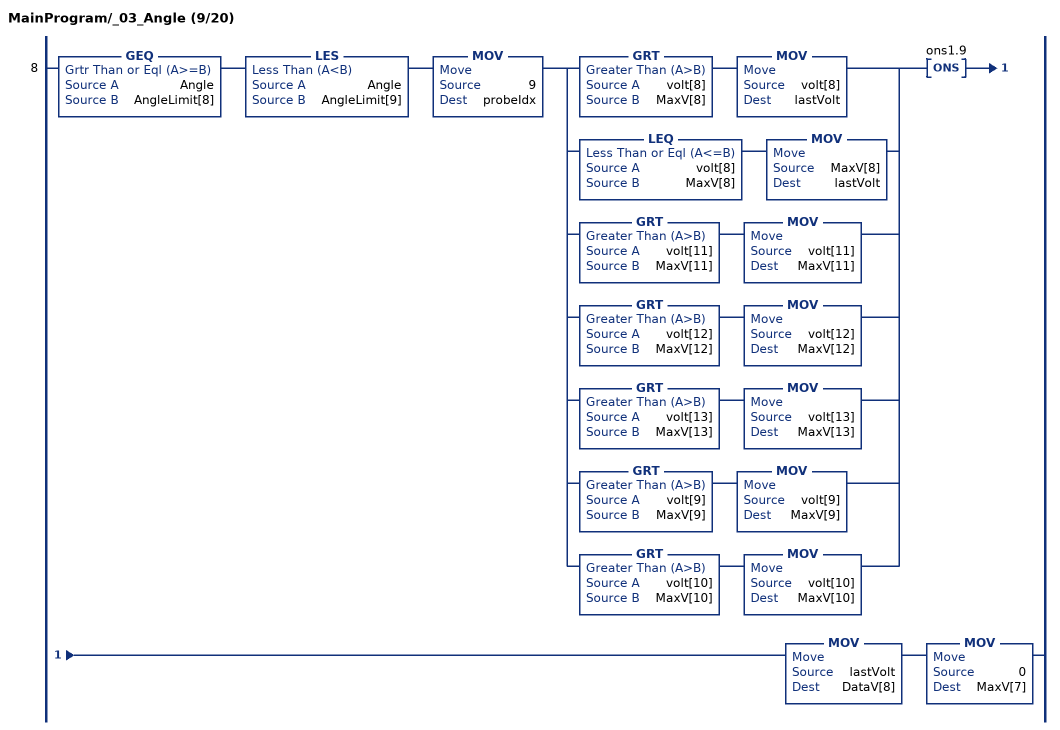
   8: GEQ(Angle,AngleLimit[8])LES(Angle,AngleLimit[9])MOV(9,probeIdx)[GRT(volt[8],MaxV[8]) MOV(volt[8],lastVolt) ,LEQ(volt[8],MaxV[8]) MOV(MaxV[8],lastVolt) ,GRT(volt[11],MaxV[11]) MOV(volt[11],MaxV[11]) ,GRT(volt[12],MaxV[12]) MOV(volt[12],MaxV[12]) ,GRT(volt[13],MaxV[13]) MOV(volt[13],MaxV[13]) ,GRT(volt[9],MaxV[9]) MOV(volt[9],MaxV[9]) ,GRT(volt[10],MaxV[10]) MOV(volt[10],MaxV[10]) ]ONS(ons1.9)MOV(lastVolt,DataV[8])MOV(0,MaxV[7]);
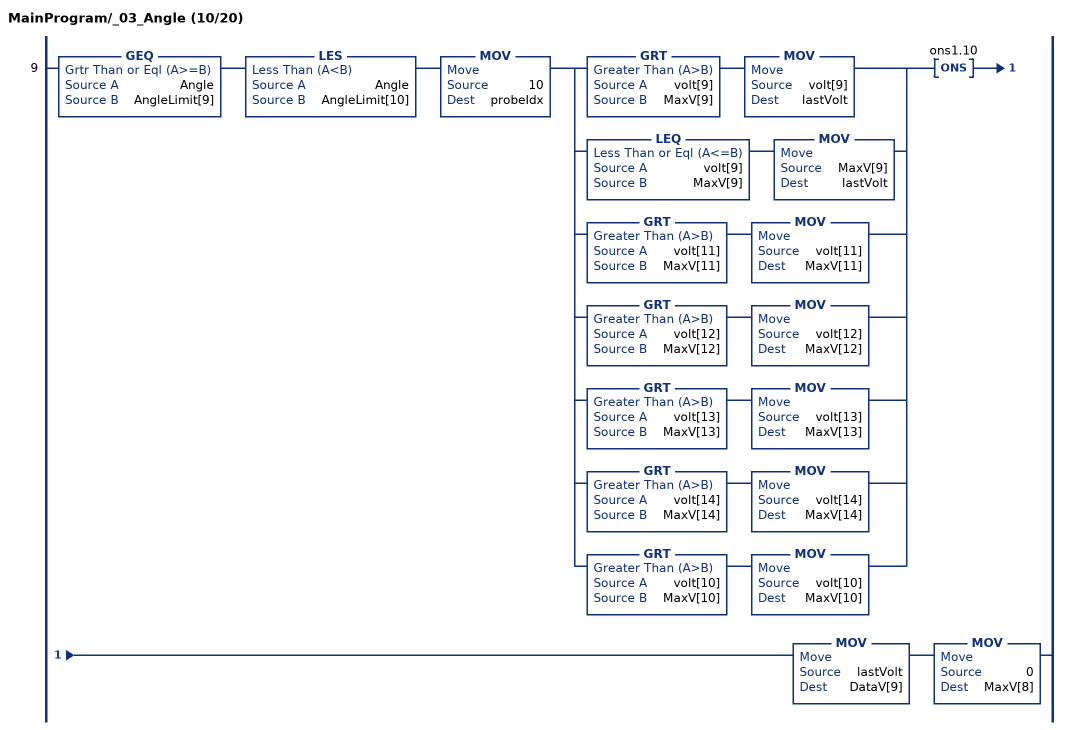
   9: GEQ(Angle,AngleLimit[9])LES(Angle,AngleLimit[10])MOV(10,probeIdx)[GRT(volt[9],MaxV[9]) MOV(volt[9],lastVolt) ,LEQ(volt[9],MaxV[9]) MOV(MaxV[9],lastVolt) ,GRT(volt[11],MaxV[11]) MOV(volt[11],MaxV[11]) ,GRT(volt[12],MaxV[12]) MOV(volt[12],MaxV[12]) ,GRT(volt[13],MaxV[13]) MOV(volt[13],MaxV[13]) ,GRT(volt[14],MaxV[14]) MOV(volt[14],MaxV[14]) ,GRT(volt[10],MaxV[10]) MOV(volt[10],MaxV[10]) ]ONS(ons1.10)MOV(lastVolt,DataV[9])MOV(0,MaxV[8]);
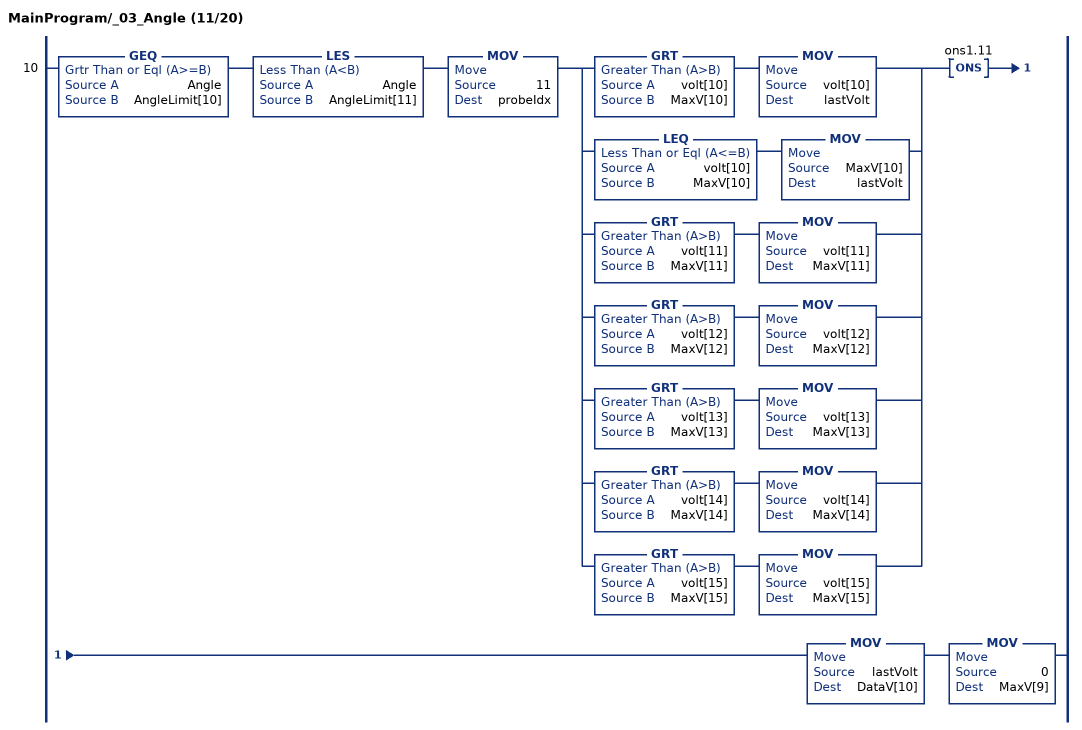
   10: GEQ(Angle,AngleLimit[10])LES(Angle,AngleLimit[11])MOV(11,probeIdx)[GRT(volt[10],MaxV[10]) MOV(volt[10],lastVolt) ,LEQ(volt[10],MaxV[10]) MOV(MaxV[10],lastVolt) ,GRT(volt[11],MaxV[11]) MOV(volt[11],MaxV[11]) ,GRT(volt[12],MaxV[12]) MOV(volt[12],MaxV[12]) ,GRT(volt[13],MaxV[13]) MOV(volt[13],MaxV[13]) ,GRT(volt[14],MaxV[14]) MOV(volt[14],MaxV[14]) ,GRT(volt[15],MaxV[15]) MOV(volt[15],MaxV[15]) ]ONS(ons1.11)MOV(lastVolt,DataV[10])MOV(0,MaxV[9]);
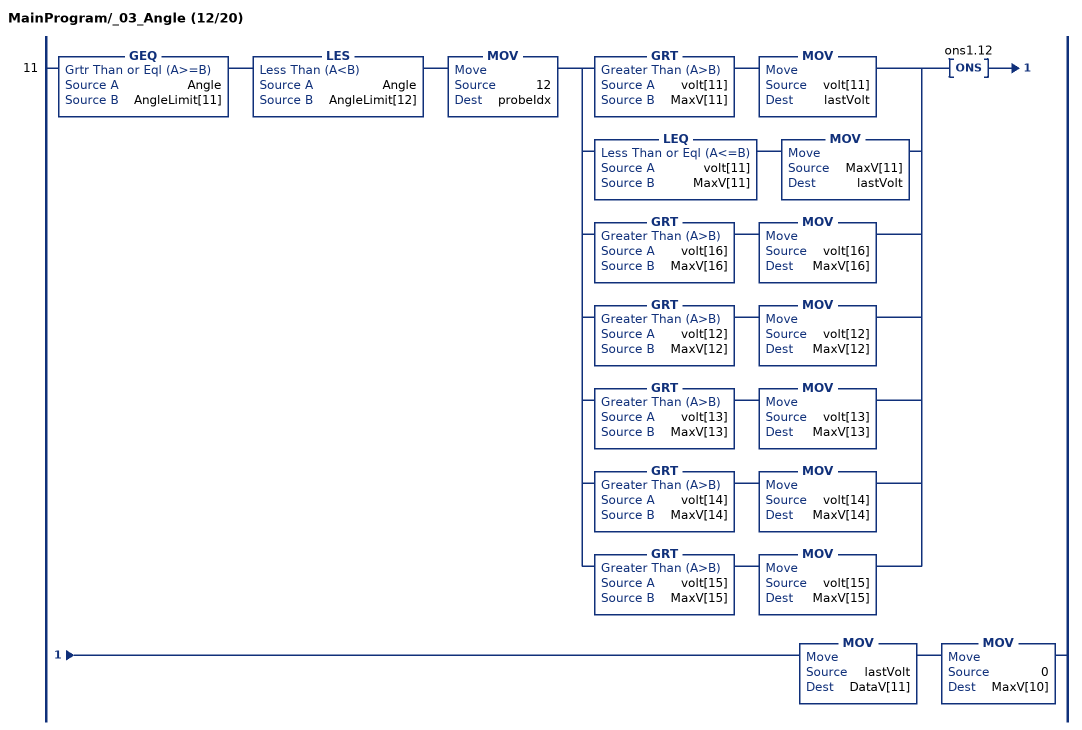
   11: GEQ(Angle,AngleLimit[11])LES(Angle,AngleLimit[12])MOV(12,probeIdx)[GRT(volt[11],MaxV[11]) MOV(volt[11],lastVolt) ,LEQ(volt[11],MaxV[11]) MOV(MaxV[11],lastVolt) ,GRT(volt[16],MaxV[16]) MOV(volt[16],MaxV[16]) ,GRT(volt[12],MaxV[12]) MOV(volt[12],MaxV[12]) ,GRT(volt[13],MaxV[13]) MOV(volt[13],MaxV[13]) ,GRT(volt[14],MaxV[14]) MOV(volt[14],MaxV[14]) ,GRT(volt[15],MaxV[15]) MOV(volt[15],MaxV[15]) ]ONS(ons1.12)MOV(lastVolt,DataV[11])MOV(0,MaxV[10]);
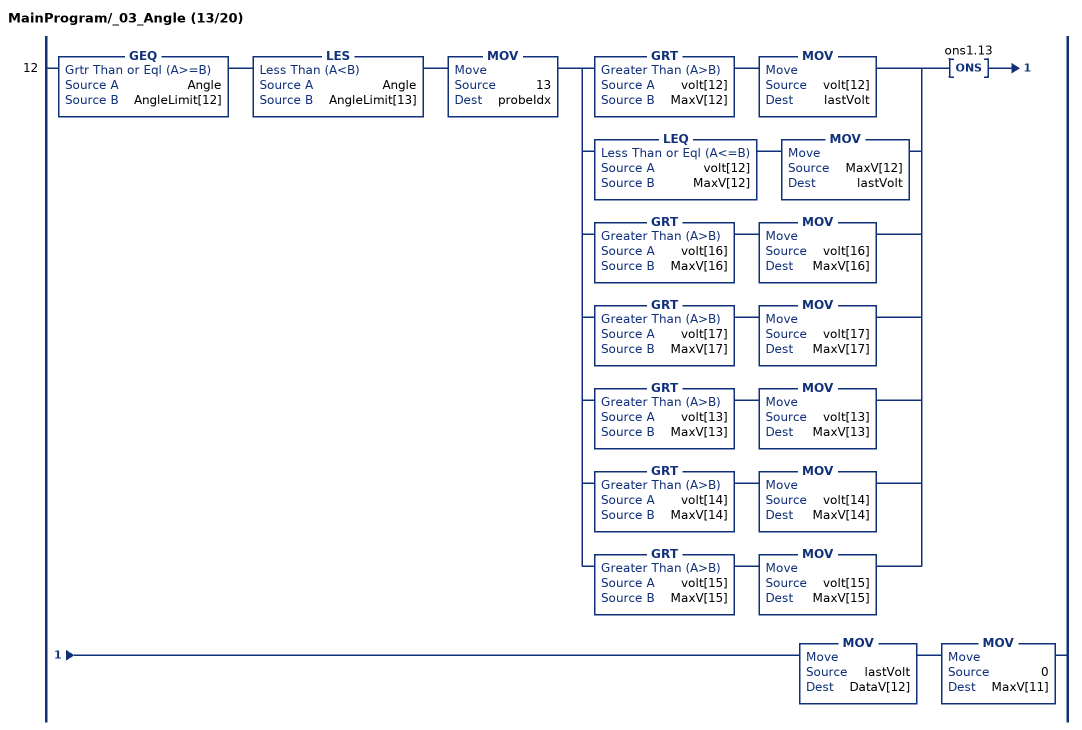
   12: GEQ(Angle,AngleLimit[12])LES(Angle,AngleLimit[13])MOV(13,probeIdx)[GRT(volt[12],MaxV[12]) MOV(volt[12],lastVolt) ,LEQ(volt[12],MaxV[12]) MOV(MaxV[12],lastVolt) ,GRT(volt[16],MaxV[16]) MOV(volt[16],MaxV[16]) ,GRT(volt[17],MaxV[17]) MOV(volt[17],MaxV[17]) ,GRT(volt[13],MaxV[13]) MOV(volt[13],MaxV[13]) ,GRT(volt[14],MaxV[14]) MOV(volt[14],MaxV[14]) ,GRT(volt[15],MaxV[15]) MOV(volt[15],MaxV[15]) ]ONS(ons1.13)MOV(lastVolt,DataV[12])MOV(0,MaxV[11]);
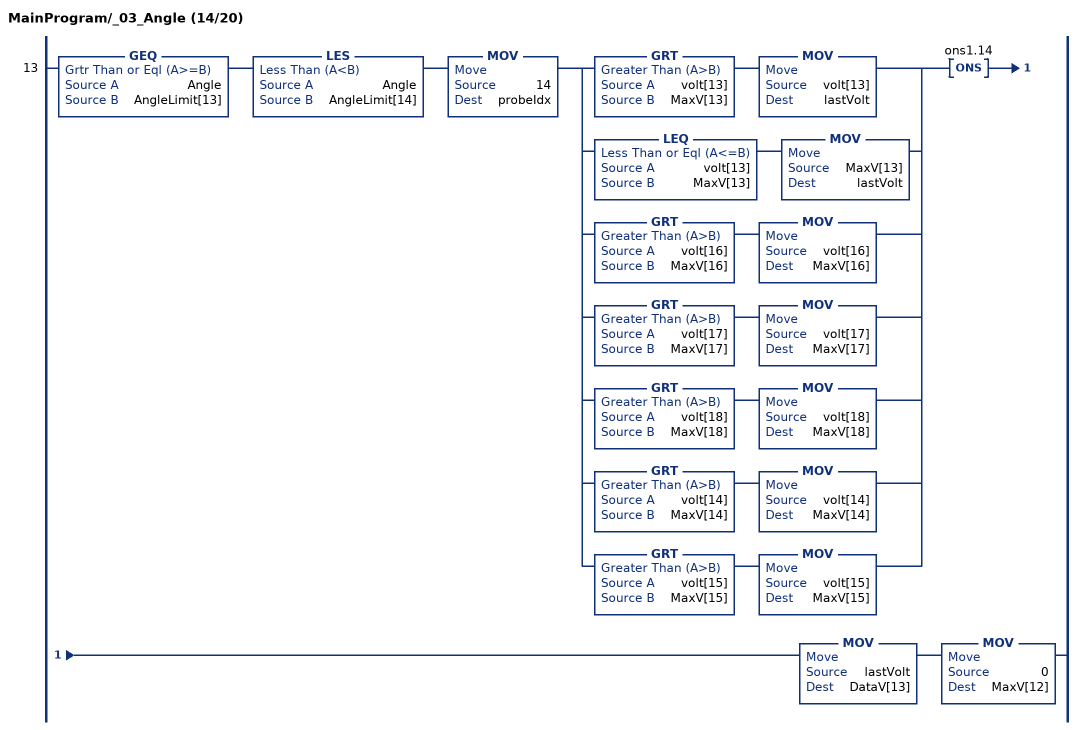
   13: GEQ(Angle,AngleLimit[13])LES(Angle,AngleLimit[14])MOV(14,probeIdx)[GRT(volt[13],MaxV[13]) MOV(volt[13],lastVolt) ,LEQ(volt[13],MaxV[13]) MOV(MaxV[13],lastVolt) ,GRT(volt[16],MaxV[16]) MOV(volt[16],MaxV[16]) ,GRT(volt[17],MaxV[17]) MOV(volt[17],MaxV[17]) ,GRT(volt[18],MaxV[18]) MOV(volt[18],MaxV[18]) ,GRT(volt[14],MaxV[14]) MOV(volt[14],MaxV[14]) ,GRT(volt[15],MaxV[15]) MOV(volt[15],MaxV[15]) ]ONS(ons1.14)MOV(lastVolt,DataV[13])MOV(0,MaxV[12]);
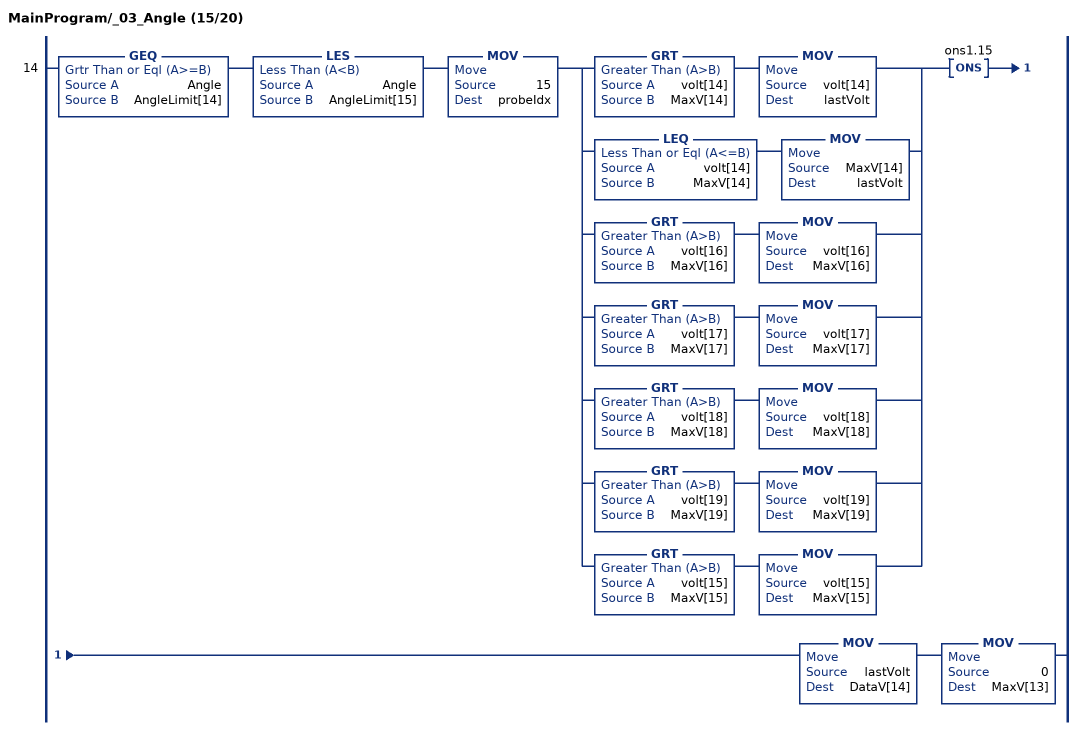
   14: GEQ(Angle,AngleLimit[14])LES(Angle,AngleLimit[15])MOV(15,probeIdx)[GRT(volt[14],MaxV[14]) MOV(volt[14],lastVolt) ,LEQ(volt[14],MaxV[14]) MOV(MaxV[14],lastVolt) ,GRT(volt[16],MaxV[16]) MOV(volt[16],MaxV[16]) ,GRT(volt[17],MaxV[17]) MOV(volt[17],MaxV[17]) ,GRT(volt[18],MaxV[18]) MOV(volt[18],MaxV[18]) ,GRT(volt[19],MaxV[19]) MOV(volt[19],MaxV[19]) ,GRT(volt[15],MaxV[15]) MOV(volt[15],MaxV[15]) ]ONS(ons1.15)MOV(lastVolt,DataV[14])MOV(0,MaxV[13]);
